FUNCTION_BLOCK POU_Auto_Trigger_Kamera

VAR_INPUT
	
		EA_Kamera_Index			: INT;
END_VAR

VAR
	
	//Locale Variablen
	L_Enable: 					BOOL;
	L_TEMP_CAM_ID: 				INT;
	L_Step_ID: 					INT := 0;
	L_SUCCESS:					BOOL;
	L_Done:						BOOL;
	L_Test_ID: 					INT := 1;
	L_Delay_TON : 				TON;
	L_Error_TON : 				TON;
	
END_VAR

IF NOT L_Enable THEN
	L_Step_ID := 0;
	RETURN;
END_IF

CASE L_Step_ID OF
	
0:
	//1. Überprüfen ob Kamera bereit ist, falls ja Trigger senden
	L_Error_TON(IN := TRUE, PT:= T#5S);
	
	L_SUCCESS := Python_Kamera_Daten.Lokal[EA_Kamera_Index].STAT.Active AND
					Python_Checker.Python_Active AND
					NOT Python_Kamera_Daten.Lokal[EA_Kamera_Index].STAT.Busy; 
	IF L_SUCCESS THEN
		Python_Kamera_Daten.Lokal[EA_Kamera_Index].CMD.ID := CONCAT('Test_', INT_TO_STRING(L_Test_ID));
		Python_Kamera_Daten.Lokal[EA_Kamera_Index].CMD.Trigger := TRUE;
		
		// Hier wird STAT von Regime
		Python_Kamera_Daten.Lokal[EA_Kamera_Index].STAT.IsDone := FALSE;
		Python_Kamera_Daten.Lokal[EA_Kamera_Index].STAT.PictureValid := FALSE;
		//
		
		L_Error_TON(IN:=FALSE);
		L_Step_ID := 10;
	END_IF
	
	IF L_Error_TON.Q THEN
		L_Error_TON(IN:=FALSE);
		L_Step_ID := 100;	
	END_IF
	
10:
	//2. Überprüfe ob das Bild valide war und ob der Auftrag abgeschlossen ist
	L_Error_TON(IN := TRUE, PT:= T#5S);
	
	L_Done :=  Python_Kamera_Daten.Lokal[EA_Kamera_Index].STAT.IsDone AND
					Python_Kamera_Daten.Lokal[EA_Kamera_Index].STAT.PictureValid AND
					NOT Python_Kamera_Daten.Lokal[EA_Kamera_Index].STAT.Busy ;
	IF L_DONE THEN
		L_Step_ID := 20;
		L_Error_TON(IN:=FALSE);
	END_IF
	
	IF L_Error_TON.Q THEN
		L_Error_TON(IN:=FALSE);
		L_Step_ID := 100;	
	END_IF

20:
	//3. Trigger zurücksetzen
	Python_Kamera_Daten.Lokal[EA_Kamera_Index].CMD.Trigger := FALSE;
	//Increase Test ID
	L_Test_ID := L_Test_ID + 1;
	IF L_Test_ID > 100 THEN
		L_Test_ID := 1;
	END_IF
	L_Step_ID := 30;
	
30:
 	//4. ein kleiner delay,sodass nur alle 2 sekunden getriggert wird
 	L_Delay_TON(IN := TRUE, PT := Parameter.Lokal[EA_Kamera_Index].Value);
	
	IF L_Delay_TON.Q THEN
		L_Delay_TON(IN:= FALSE);
		L_Step_ID := 0;
	END_IF
	
100:
	L_Enable := FALSE;
	Python_Checker.Python_ERROR := TRUE;
	
	
	
	

END_CASE

END_FUNCTION_BLOCK

(* stored: Version 1.1.0.1, ProductVersion 3.1.4024.12
   POU POU_Auto_Trigger_Kamera: Id {7ddd821b-b727-42f6-bcf5-efed6bb16a7f}, SpecialFunc None *)
